FUNCTION_BLOCK SS3_ifb_ps_Axis (* Composite FB wrapping other FBs *)
  (* Standard: 61499-2 *)
  (* Version 1.0, 2025-05-26, PS_Transformer_for_Unknown *)
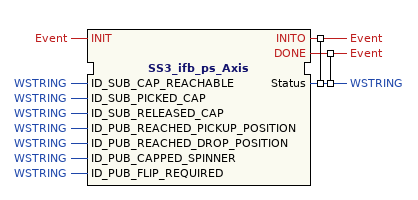
  EVENT_INPUT
    INIT; (* Initialization Request *)
  END_EVENT
  EVENT_OUTPUT
    INITO WITH Status; (* Initialization Confirm *)
    DONE WITH Status; (* Execution Confirmation *)
  END_EVENT
  VAR_INPUT
    ID_SUB_CAP_REACHABLE : WSTRING;
    ID_SUB_PICKED_CAP : WSTRING;
    ID_SUB_RELEASED_CAP : WSTRING;
    ID_PUB_REACHED_PICKUP_POSITION : WSTRING;
    ID_PUB_REACHED_DROP_POSITION : WSTRING;
    ID_PUB_CAPPED_SPINNER : WSTRING;
    ID_PUB_FLIP_REQUIRED : WSTRING;
  END_VAR
  VAR_OUTPUT
    Status : WSTRING; (* Output event qualifier *)
  END_VAR
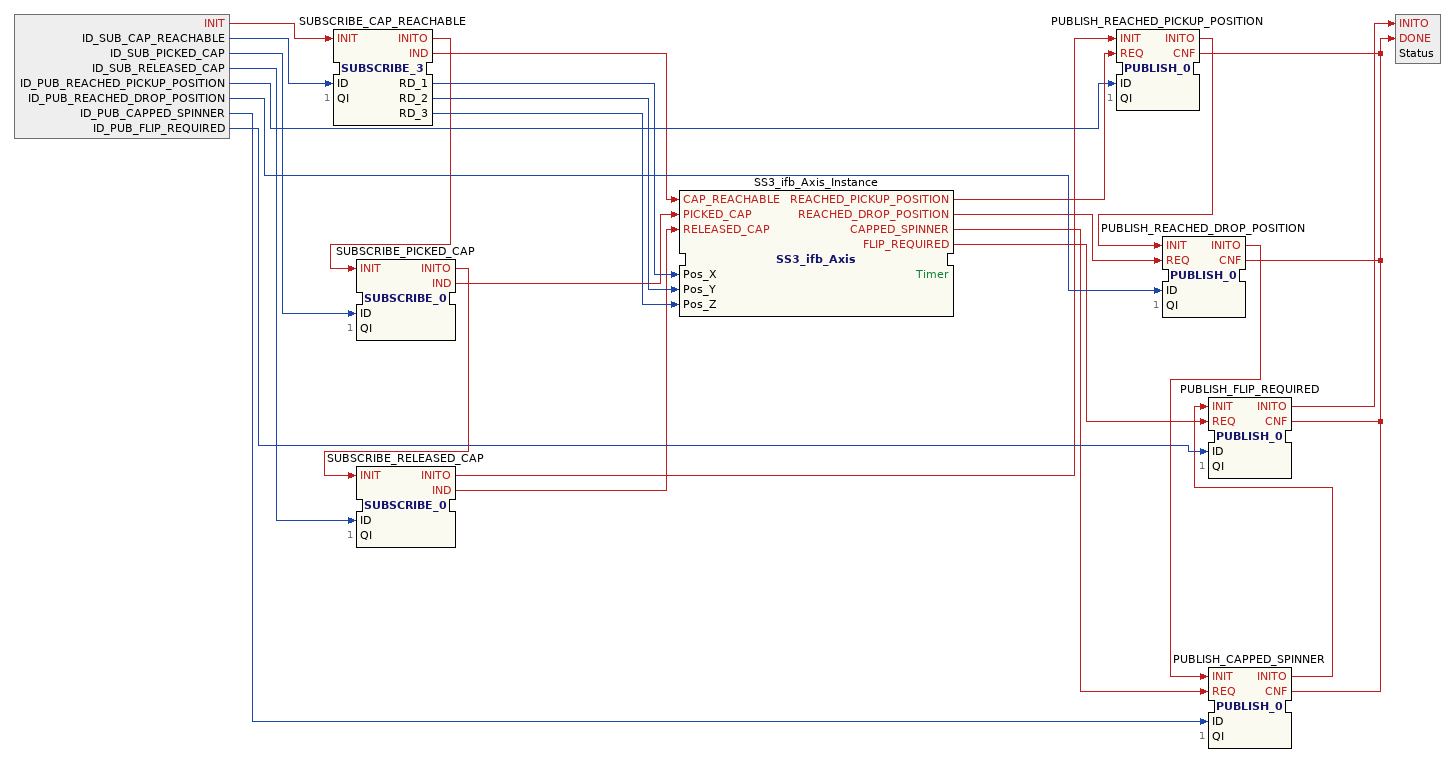
  FBS
    SS3_ifb_Axis_Instance : SS3_ifb_Axis;
    SUBSCRIBE_CAP_REACHABLE : SUBSCRIBE_3(QI := 1);
    SUBSCRIBE_PICKED_CAP : SUBSCRIBE_0(QI := 1);
    SUBSCRIBE_RELEASED_CAP : SUBSCRIBE_0(QI := 1);
    PUBLISH_REACHED_PICKUP_POSITION : PUBLISH_0(QI := 1);
    PUBLISH_REACHED_DROP_POSITION : PUBLISH_0(QI := 1);
    PUBLISH_CAPPED_SPINNER : PUBLISH_0(QI := 1);
    PUBLISH_FLIP_REQUIRED : PUBLISH_0(QI := 1);
  END_FBS
  EVENT_CONNECTIONS
    INIT TO SUBSCRIBE_CAP_REACHABLE.INIT;
    SUBSCRIBE_CAP_REACHABLE.INITO TO SUBSCRIBE_PICKED_CAP.INIT;
    SUBSCRIBE_PICKED_CAP.INITO TO SUBSCRIBE_RELEASED_CAP.INIT;
    SUBSCRIBE_RELEASED_CAP.INITO TO PUBLISH_REACHED_PICKUP_POSITION.INIT;
    PUBLISH_REACHED_PICKUP_POSITION.INITO TO PUBLISH_REACHED_DROP_POSITION.INIT;
    PUBLISH_REACHED_DROP_POSITION.INITO TO PUBLISH_CAPPED_SPINNER.INIT;
    PUBLISH_CAPPED_SPINNER.INITO TO PUBLISH_FLIP_REQUIRED.INIT;
    PUBLISH_FLIP_REQUIRED.INITO TO INITO;
    SUBSCRIBE_CAP_REACHABLE.IND TO SS3_ifb_Axis_Instance.CAP_REACHABLE;
    SUBSCRIBE_PICKED_CAP.IND TO SS3_ifb_Axis_Instance.PICKED_CAP;
    SUBSCRIBE_RELEASED_CAP.IND TO SS3_ifb_Axis_Instance.RELEASED_CAP;
    SS3_ifb_Axis_Instance.REACHED_PICKUP_POSITION TO PUBLISH_REACHED_PICKUP_POSITION.REQ;
    SS3_ifb_Axis_Instance.REACHED_DROP_POSITION TO PUBLISH_REACHED_DROP_POSITION.REQ;
    SS3_ifb_Axis_Instance.CAPPED_SPINNER TO PUBLISH_CAPPED_SPINNER.REQ;
    SS3_ifb_Axis_Instance.FLIP_REQUIRED TO PUBLISH_FLIP_REQUIRED.REQ;
    PUBLISH_REACHED_PICKUP_POSITION.CNF TO DONE;
    PUBLISH_REACHED_DROP_POSITION.CNF TO DONE;
    PUBLISH_CAPPED_SPINNER.CNF TO DONE;
    PUBLISH_FLIP_REQUIRED.CNF TO DONE;
  END_CONNECTIONS
  DATA_CONNECTIONS
    ID_SUB_CAP_REACHABLE TO SUBSCRIBE_CAP_REACHABLE.ID;
    ID_SUB_PICKED_CAP TO SUBSCRIBE_PICKED_CAP.ID;
    ID_SUB_RELEASED_CAP TO SUBSCRIBE_RELEASED_CAP.ID;
    ID_PUB_REACHED_PICKUP_POSITION TO PUBLISH_REACHED_PICKUP_POSITION.ID;
    ID_PUB_REACHED_DROP_POSITION TO PUBLISH_REACHED_DROP_POSITION.ID;
    ID_PUB_CAPPED_SPINNER TO PUBLISH_CAPPED_SPINNER.ID;
    ID_PUB_FLIP_REQUIRED TO PUBLISH_FLIP_REQUIRED.ID;
    SUBSCRIBE_CAP_REACHABLE.RD_1 TO SS3_ifb_Axis_Instance.Pos_X;
    SUBSCRIBE_CAP_REACHABLE.RD_2 TO SS3_ifb_Axis_Instance.Pos_Y;
    SUBSCRIBE_CAP_REACHABLE.RD_3 TO SS3_ifb_Axis_Instance.Pos_Z;
  END_CONNECTIONS
END_FUNCTION_BLOCK
